FUNCTION_BLOCK Dictionary_TestSuite EXTENDS TcUnit.FB_TestSuite
VAR
END_VAR

CheckAddOrUpdateCorrectlyAddsNewKey();
CheckAddOrUpdateCorrectlyUpdatesExistingKey();
CheckClear();
CheckContainsKeyIsFalse();
CheckContainsKeyIsTrue();
CheckCount();
CheckEnumeratorIsInvalidAfterChange();
CheckGetEnumerator();
CheckGetKeysReturnsACollection();
CheckGetKeysReturnsACollectionOfValidKeys();
CheckOffEvent();
CheckOnceEvent();
CheckOnChangedEvent();
CheckOnDisposedEvent();
CheckRemoveExisting();
CheckRemoveNonExisting();
CheckTryAddCorrectlyAddsNewKey();
CheckTryAddCorrectlyIgnoresUpdateWhenDuplicateFound();
CheckTryAddCorrectlyReturnsFalseWhenDuplicateFound();
CheckTryAddCorrectlyReturnsTrueWhenAddNewKey();
CheckTryGetValueTo();
CheckTryGetValue();
CheckWorksWithArrays();
CheckWorksWithIntegers();
CheckWorksWithStrings();
CheckIsEmptyWhenEmpty();
CheckIsEmptyWhenFull();

METHOD PUBLIC CheckAddOrUpdateCorrectlyAddsNewKey
VAR
	in : INT := 123;
	out : INT;
	expected : INT := 123;
	dictionary : Dictionary;
END_VAR
TEST('CheckAddOrUpdateCorrectlyAddsNewKey');

dictionary.AddOrUpdate('a',in);
dictionary.TryGetValue('a',out);

AssertEquals(
	Expected := expected,
	Actual := out,
	Message := 'Did not produce the expected result'
);

TEST_FINISHED();
END_METHOD

METHOD PUBLIC CheckAddOrUpdateCorrectlyUpdatesExistingKey
VAR
	in1 : INT := 123;
	in2 : INT := 456;
	out : INT;
	expected : INT := 456;
	dictionary : Dictionary;
END_VAR
TEST('CheckAddOrUpdateCorrectlyUpdatesExistingKey');

dictionary.AddOrUpdate('a',in1);
dictionary.AddOrUpdate('a',in2);
dictionary.TryGetValue('a',out);

AssertEquals(
	Expected := expected,
	Actual := out,
	Message := 'Did not produce the expected result'
);

TEST_FINISHED();
END_METHOD

METHOD PUBLIC CheckClear
VAR
	in1 : INT := 123;
	in2 : INT := 456;
	out : INT;
	expected : INT := 456;
	dictionary : Dictionary;
END_VAR
TEST('CheckClear');

dictionary.TryAdd('a',in1);
dictionary.Clear();
dictionary.TryAdd('a',in2); // if the dictionary was not empty then this would fail.
dictionary.TryGetValue('a',out);

// @TEST-ASSSERT
AssertEquals(
	Expected := expected,
	Actual := out,
	Message := 'Did not produce the expected result'
);

TEST_FINISHED();
END_METHOD

METHOD PUBLIC CheckContainsKeyIsFalse
VAR
	in1 : INT := 123;
	in2 : INT := 456;
	in3 : INT := 789;
	result : BOOL;
	dictionary : Dictionary;
END_VAR
TEST('CheckContainsKeyIsFalse');

dictionary.TryAdd('a',in1);
dictionary.TryAdd('b',in2);
dictionary.TryAdd('c',in3);

result := dictionary.ContainsKey('d');

AssertFalse(
	Condition := result,
	Message := 'Did not produce the expected result'
);

TEST_FINISHED();
END_METHOD

METHOD PUBLIC CheckContainsKeyIsTrue
VAR
	in1 : INT := 123;
	in2 : INT := 456;
	in3 : INT := 789;
	result : BOOL;
	dictionary : Dictionary;
END_VAR
TEST('CheckContainsKeyIsTrue');

dictionary.TryAdd('a',in1);
dictionary.TryAdd('b',in2);
dictionary.TryAdd('c',in3);

result := dictionary.ContainsKey('b');

AssertTrue(
	Condition := result,
	Message := 'Did not produce the expected result'
);

TEST_FINISHED();
END_METHOD

METHOD PUBLIC CheckCount
VAR
	in1 : INT := 123;
	in2 : INT := 456;
	in3 : INT := 789;
	out : DINT;
	expected : DINT := 3;
	dictionary : Dictionary;
END_VAR
TEST('CheckCount');

dictionary.TryAdd('a',in1);
dictionary.TryAdd('b',in2);
dictionary.TryAdd('c',in3);
out := dictionary.Count;

AssertEquals(
	Expected := expected,
	Actual := out,
	Message := 'Did not produce the expected result'
);

TEST_FINISHED();
END_METHOD

METHOD PUBLIC CheckEnumeratorIsInvalidAfterChange
VAR
	in : INT := 123;
	result : BOOL;
	dictionary : Dictionary;
	enumerator : I_ForwardEnumerator;
END_VAR
TEST('CheckEnumeratorIsInvalidAfterChange');

enumerator := dictionary.GetEnumerator();
dictionary.TryAdd('a',in);

result := enumerator.IsValid;
enumerator.Dispose();

AssertFalse(
	Condition := result,
	Message := 'Method returned true'
);

TEST_FINISHED();
END_METHOD

METHOD PUBLIC CheckGetEnumerator
VAR
	enumerator : I_ForwardEnumerator;
	dictionary : Dictionary;
END_VAR
TEST('CheckGetEnumerator');

enumerator := dictionary.GetEnumerator();

AssertTrue(
	Condition := (enumerator <> 0),
	Message := 'Did not return an enumerator'
);

enumerator.Dispose();

TEST_FINISHED();
END_METHOD

METHOD PUBLIC CheckGetKeysReturnsACollection
VAR
	result : BOOL;
	dictionary : Dictionary;
	collection : I_Collection;
END_VAR
TEST('CheckGetKeysReturnsACollection');

collection := dictionary.GetKeys();

result := collection <> 0;

IF result THEN
	collection.Dispose();
END_IF

AssertTrue(
	Condition := result,
	Message := 'Did not produce the expected result'
);

TEST_FINISHED();
END_METHOD

METHOD PUBLIC CheckGetKeysReturnsACollectionOfValidKeys
VAR
	in1 : INT := 123;
	in2 : INT := 456;
	in3 : INT := 789;
	out : ARRAY [0..2] OF T_MAXSTRING;
	expected : ARRAY [0..2] OF T_MAXSTRING;
	result,resulta,resultb,resultc : BOOL;
	dictionary : Dictionary;
	collection : I_Collection;
END_VAR
TEST('CheckGetKeysReturnsACollectionOfValidKeys');

// clear the out and expected variables as strings may contain left over data
memset(ADR(out),0,SIZEOF(out));
memset(ADR(expected),0,SIZEOF(expected));

// now create the "expected"
expected[0] := 'a';
expected[1] := 'b';
expected[2] := 'c';

// now setup the test
dictionary.TryAdd('a',in1);
dictionary.TryAdd('b',in2);
dictionary.TryAdd('c',in3);

collection := dictionary.GetKeys();
collection.TryCopyTo(out);
collection.Dispose();

// create the test result
resulta := expected[0] = out[0];
resultb := expected[1] = out[1];
resultc := expected[2] = out[2];
result := resulta AND resultb AND resultc;

AssertTrue(
	Condition := result,
	Message := 'Did not return an enumerator'
);

TEST_FINISHED();
END_METHOD

METHOD PUBLIC CheckIsEmptyWhenEmpty
VAR
	result : BOOL;
	dictionary : Dictionary;
END_VAR
TEST('CheckIsEmptyWhenEmpty');

// @TEST-RUN
result := dictionary.IsEmpty;

// @TEST-ASSSERT
AssertTrue(
	Condition := result,
	Message := 'Incorrect state of IsEmpty'
);

TEST_FINISHED();
END_METHOD

METHOD PUBLIC CheckIsEmptyWhenFull
VAR
	in : INT := 123;
	result : BOOL;
	dictionary : Dictionary;
END_VAR
TEST('CheckIsEmptyWhenFull');

// @TEST-FIXTURE
dictionary.AddOrUpdate('a',in);

// @TEST-RUN
result := dictionary.IsEmpty;

// @TEST-ASSSERT
AssertFalse(
	Condition := result,
	Message := 'Incorrect state of IsEmpty'
);

TEST_FINISHED();
END_METHOD

METHOD PUBLIC CheckOffEvent
VAR
	value : INT := 123;
	dictionary : Dictionary;
	handler : KeyValueCollectionChangedEventHandler(ExpectedOriginator := dictionary);
END_VAR
TEST('CheckOffEvent');

dictionary.OnEvent('OnChanged',handler);
dictionary.OffEvent('OnChanged',handler);

dictionary.TryAdd('a',value);

AssertFalse(
	Condition := handler.EventReceived,
	Message := 'OnceEvent emitted the OnChanged event more than once'
);

TEST_FINISHED();
END_METHOD

METHOD PUBLIC CheckOnceEvent
VAR
	value : INT := 123;
	dictionary : Dictionary;
	handler : KeyValueCollectionChangedEventHandler(ExpectedOriginator := dictionary);
END_VAR
TEST('CheckOnceEvent');

dictionary.OnceEvent('OnChanged',handler);
dictionary.TryAdd('a',value);
handler.Reset();

dictionary.TryAdd('a',value);

AssertFalse(
	Condition := handler.EventReceived,
	Message := 'OnceEvent emitted the OnChanged event more than once'
);

TEST_FINISHED();
END_METHOD

METHOD PUBLIC CheckOnChangedEvent
VAR
	value : INT := 123;
	dictionary : Dictionary;
	handler : KeyValueCollectionChangedEventHandler(ExpectedOriginator := dictionary);
END_VAR
TEST('CheckOnChangedEvent');

dictionary.OnEvent('OnChanged', handler);
dictionary.TryAdd('a',value);

AssertTrue(
	Condition := handler.EventReceived,
	Message := 'Did not emit the OnChanged event'
);

AssertTrue(
	Condition := handler.FromExpectedOriginator,
	Message := 'Did not include itself in the OnChanged event'
);

TEST_FINISHED();
END_METHOD

METHOD PUBLIC CheckOnDisposedEvent
VAR
	value : INT := 123;
	pDictionary : POINTER TO Dictionary;
	handler : KeyValueCollectionDisposedEventHandler(ExpectedOriginator := 0);
END_VAR
TEST('CheckOnDisposedEvent');

pDictionary := __NEW(Dictionary);
handler.SetExpectedOriginator(pDictionary^);
pDictionary^.OnEvent('OnDisposed', handler);

pDictionary^.Dispose();

AssertTrue(
	Condition := handler.EventReceived,
	Message := 'Did not emit the OnDisposed event'
);

AssertTrue(
	Condition := handler.FromExpectedOriginator,
	Message := 'Did not include itself in the OnDisposed event'
);

TEST_FINISHED();
END_METHOD

METHOD PRIVATE CheckRemoveExisting
VAR
	in1 : INT := 123;
	in2 : INT := 456;
	in3 : INT := 789;
	result : BOOL;
	dictionary : Dictionary;
END_VAR
TEST('CheckRemoveExisting');

dictionary.TryAdd('a',in1);
dictionary.TryAdd('b',in2);
dictionary.TryAdd('c',in3);

dictionary.Remove('c');

result := dictionary.ContainsKey('c');

AssertFalse(
	Condition := result,
	Message := 'Did not produce the expected result'
);

TEST_FINISHED();
END_METHOD

METHOD PRIVATE CheckRemoveNonExisting
VAR
	in1 : INT := 123;
	in2 : INT := 456;
	in3 : INT := 789;
	out : DINT;
	expected : DINT := 3;
	dictionary : Dictionary;
END_VAR
TEST('CheckRemoveNonExisting');

dictionary.TryAdd('a',in1);
dictionary.TryAdd('b',in2);
dictionary.TryAdd('c',in3);

dictionary.Remove('d');

out := dictionary.Count;

AssertEquals(
	Expected := expected,
	Actual := out,
	Message := 'Did not produce the expected result'
);

TEST_FINISHED();
END_METHOD

METHOD PUBLIC CheckTryAddCorrectlyAddsNewKey
VAR
	in : INT := 123;
	out : INT;
	expected : INT := 123;
	dictionary : Dictionary;
END_VAR
TEST('CheckTryAddCorrectlyAddsNewKey');

dictionary.TryAdd('a',in);
dictionary.TryGetValue('a',out);

AssertEquals(
	Expected := expected,
	Actual := out,
	Message := 'Did not produce the expected result'
);

TEST_FINISHED();
END_METHOD

METHOD PUBLIC CheckTryAddCorrectlyIgnoresUpdateWhenDuplicateFound
VAR
	in1 : INT := 123;
	in2 : INT := 456;
	out : INT;
	expected : INT := 123;
	result : BOOL;
	dictionary : Dictionary;
END_VAR
TEST('CheckTryAddCorrectlyIgnoresUpdateWhenDuplicateFound');

dictionary.TryAdd('a',in1);
dictionary.TryAdd('a',in2);
dictionary.TryGetValue('a',out);

AssertEquals(
	Expected := expected,
	Actual := out,
	Message := 'Did not produce the expected result'
);

TEST_FINISHED();
END_METHOD

METHOD PUBLIC CheckTryAddCorrectlyReturnsFalseWhenDuplicateFound
VAR
	in1 : INT := 123;
	in2 : INT := 456;
	result : BOOL;
	dictionary : Dictionary;
END_VAR
TEST('CheckTryAddCorrectlyReturnsFalseWhenDuplicateFound');

dictionary.TryAdd('a',in1);
result := dictionary.TryAdd('a',in2);

AssertFalse(
	Condition := result,
	Message := 'Did not produce the expected result'
);

TEST_FINISHED();
END_METHOD

METHOD PUBLIC CheckTryAddCorrectlyReturnsTrueWhenAddNewKey
VAR
	in : INT := 123;
	result : BOOL;
	dictionary : Dictionary;
END_VAR
TEST('CheckTryAddCorrectlyReturnsTrueWhenAddNewKey');

result := dictionary.TryAdd('a',in);

AssertTrue(
	Condition := result,
	Message := 'Did not produce the expected result'
);

TEST_FINISHED();
END_METHOD

METHOD PUBLIC CheckTryGetValue
VAR
	in : INT := 123;
	out : INT;
	expected : INT := 123;
	dictionary : Dictionary;
END_VAR
TEST('CheckTryGetValue');

dictionary.AddOrUpdate('a',in);
dictionary.TryGetValue('a',out);

AssertEquals(
	Expected := expected,
	Actual := out,
	Message := 'Did not produce the expected result'
);

TEST_FINISHED();
END_METHOD

METHOD PUBLIC CheckTryGetValueTo
VAR
	in : INT := 123;
	out : INT;
	expected : INT := 123;
	dictionary : Dictionary;
END_VAR
TEST('CheckTryGetValueTo');

dictionary.AddOrUpdate('a',in);
dictionary.TryGetValueTo('a',ADR(out),SIZEOF(out));

AssertEquals(
	Expected := expected,
	Actual := out,
	Message := 'Did not produce the expected result'
);

TEST_FINISHED();
END_METHOD

METHOD PUBLIC CheckWorksWithArrays
VAR
	in : ARRAY [0..1] OF REAL := [0.1,2.3];
	out : ARRAY [0..1] OF REAL;
	expected : ARRAY [0..1] OF REAL := [0.1,2.3];
	dictionary : Dictionary;
END_VAR
TEST('CheckWorksWithArrays');

dictionary.TryAdd('a',in);
dictionary.TryGetValue('a',out);

AssertEquals(
	Expected := expected,
	Actual := out,
	Message := 'Did not produce the expected result'
);

TEST_FINISHED();
END_METHOD

METHOD PUBLIC CheckWorksWithIntegers
VAR
	in : INT := 123;
	out : INT;
	expected : INT := 123;
	dictionary : Dictionary;
END_VAR
TEST('CheckWorksWithIntegers');

dictionary.TryAdd('a',in);
dictionary.TryGetValue('a',out);

AssertEquals(
	Expected := expected,
	Actual := out,
	Message := 'Did not produce the expected result'
);

TEST_FINISHED();
END_METHOD

METHOD PUBLIC CheckWorksWithStrings
VAR
	in : STRING := 'test';
	out : STRING;
	expected : STRING := 'test';
	dictionary : Dictionary;
END_VAR
TEST('CheckWorksWithStrings');

dictionary.TryAdd('a',in);
dictionary.TryGetValue('a',out);

AssertEquals(
	Expected := expected,
	Actual := out,
	Message := 'Did not produce the expected result'
);

TEST_FINISHED();
END_METHOD

END_FUNCTION_BLOCK

(* stored: Version 1.1.0.1, ProductVersion 3.1.4024.12
   POU Dictionary_TestSuite: Id {6dd685da-a543-00aa-14e8-1b871a063fb7}, SpecialFunc None
   Method CheckAddOrUpdateCorrectlyAddsNewKey: Id {4a5e823a-6418-0549-38c4-799d6345f9af}
   Method CheckAddOrUpdateCorrectlyUpdatesExistingKey: Id {9a83afdd-866e-08e8-10c1-ce5154773c53}
   Method CheckClear: Id {c97ba217-487f-06a2-137a-0f27aac18860}
   Method CheckContainsKeyIsFalse: Id {cc9a553f-1a05-0730-1dc4-cc08fa48aa1c}
   Method CheckContainsKeyIsTrue: Id {1aded3cb-0b33-0ccc-1ae5-c497bbcac1bd}
   Method CheckCount: Id {e712680b-98e8-0883-100e-3ceb234f340a}
   Method CheckEnumeratorIsInvalidAfterChange: Id {8bb7642c-819a-0267-1cd4-3712c7efefb0}
   Method CheckGetEnumerator: Id {825248e0-f3a7-03db-1742-bbe630aa8954}
   Method CheckGetKeysReturnsACollection: Id {4f41e7cb-abee-0dce-0e51-9da3592324c5}
   Method CheckGetKeysReturnsACollectionOfValidKeys: Id {bf9c5c97-1faf-02e1-090d-93cbf4034b9a}
   Method CheckIsEmptyWhenEmpty: Id {c2fb321c-ba45-061d-1d89-054aae60cad8}
   Method CheckIsEmptyWhenFull: Id {555017f9-a4e8-07e9-12f0-13b3fb8c8fac}
   Method CheckOffEvent: Id {58274f09-e5aa-0700-3dde-0a818233e28f}
   Method CheckOnceEvent: Id {a94c0486-1292-0536-2008-ec71d30b00a4}
   Method CheckOnChangedEvent: Id {7b8fa736-2926-061e-0509-3fab8e9f86a2}
   Method CheckOnDisposedEvent: Id {4624cead-2d88-0b8b-131f-f13e4c7580f7}
   Method CheckRemoveExisting: Id {82edeada-7b9b-0993-2235-161bb655d6ab}
   Method CheckRemoveNonExisting: Id {642554fd-2b01-07a0-005c-f908f549881f}
   Method CheckTryAddCorrectlyAddsNewKey: Id {15d25fe5-5915-09bf-3d0e-ab95c645cd3c}
   Method CheckTryAddCorrectlyIgnoresUpdateWhenDuplicateFound: Id {b906ba2e-1c54-0287-067a-72852533863a}
   Method CheckTryAddCorrectlyReturnsFalseWhenDuplicateFound: Id {2c51d8c9-0818-08df-275b-bc51f84570bf}
   Method CheckTryAddCorrectlyReturnsTrueWhenAddNewKey: Id {3b760531-a7f5-0c39-0f66-3928a1ad6910}
   Method CheckTryGetValue: Id {b222690f-f631-0dcd-2d72-a869546ed356}
   Method CheckTryGetValueTo: Id {a3511342-3a7d-05e0-22e5-a00aa5c4a537}
   Method CheckWorksWithArrays: Id {7e8d7f32-0c4d-0914-15c3-0e226a13243b}
   Method CheckWorksWithIntegers: Id {54206d3f-096c-0a9c-08fb-991c5d99371e}
   Method CheckWorksWithStrings: Id {67c59906-d985-0746-24fc-dd41969bd704} *)
